ABB RobotStudio station: PR15CintasInteligentesEnunciado.rspag

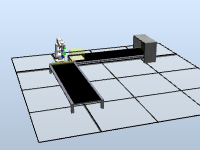
--- station ---
Station Station (saved by RobotStudio 6.5.7392.129)
Controller Sistema3
  mechanical unit ROB_1: IRB120_3_58__01, 6 joints, base frame (0, 0, 0) mm
Layout (positions relative to the parent item):
  - IRB120_3_58__01 [mechanism, from Robots\IRB120_3_58_G_01.rslib] at (0, 0, 0) mm; joint values [0, 0, 0, 0, 1.5708, 0] (rad or m)
  - SC_VentosaD50 [smart component] at (302, 0, 558) mm, rotated rx 180 ry 0 rz 180 deg
      signals: DI ElecVenturiVacio, DO ContactoVacuostato
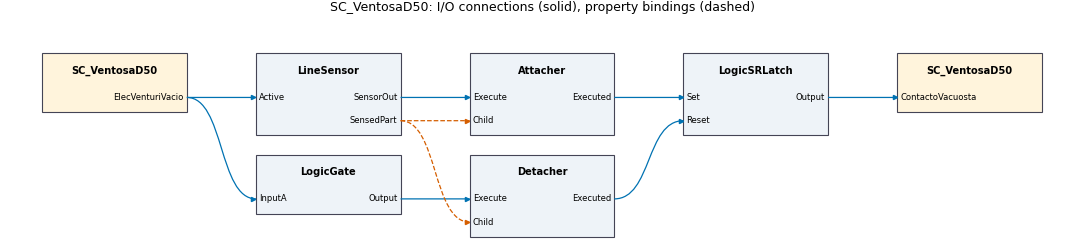
      connections:
        SC_VentosaD50.ElecVenturiVacio -> LineSensor.Active
        LineSensor.SensorOut -> Attacher.Execute
        Attacher.Executed -> LogicSRLatch.Set
        LogicSRLatch.Output -> SC_VentosaD50.ContactoVacuostato
        SC_VentosaD50.ElecVenturiVacio -> LogicGate.InputA
        LogicGate.Output -> Detacher.Execute
        Detacher.Executed -> LogicSRLatch.Reset
        LineSensor.SensedPart => Attacher.Child
        LineSensor.SensedPart => Detacher.Child
    - ToolVentosaD50 [mechanism] at (0, 0, 0) mm
        TCP TCP_ToolVentosaD50 at (0, 0, 129.5) mm
        links: VentosaCompletaD50
    - Attacher [smart component, from Components\Attacher.rslib]
        properties: Parent=ToolVentosaD50; Flange=0; Child=(none); Mount=false; Offset=[0 0 0]; Orientation=[0 0 0]
    - Detacher [smart component, from Components\Detacher.rslib]
        properties: Child=(none); KeepPosition=true
    - LineSensor [smart component, from Components\LineSensor.rslib] at (0, 0, 126) mm
        properties: Start=[0 0 0]; End=[0 0 0.015]; Radius=0.001; SensedPart=(none); SensedPoint=[3.0517578125E-08 0.427339996337891 0.290037750244141]
      - _sensorPart_ [part]
    - LogicGate [smart component, from Components\LogicGate.rslib]
        properties: Operator=NOT; Delay=0
    - LogicSRLatch [smart component, from Components\LogicSRLatch.rslib]
  - SC_CintaTransportadoraAlimentador [smart component] at (250, -300, 0) mm
      signals: DI diMotorCinta, DO doSensorCajas
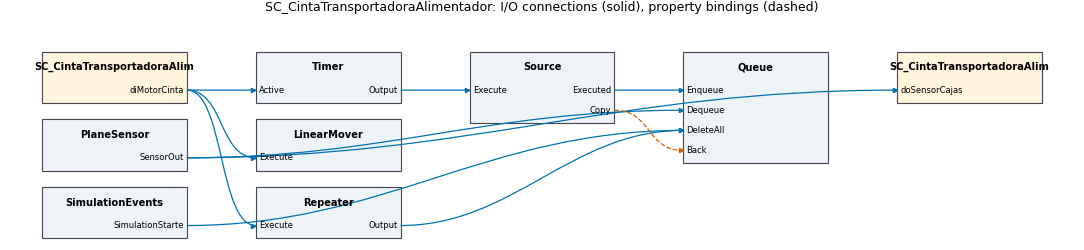
      connections:
        SC_CintaTransportadoraAlimentador.diMotorCinta -> Timer.Active
        SC_CintaTransportadoraAlimentador.diMotorCinta -> LinearMover.Execute
        Timer.Output -> Source.Execute
        Source.Executed -> Queue.Enqueue
        PlaneSensor.SensorOut -> Queue.Dequeue
        PlaneSensor.SensorOut -> SC_CintaTransportadoraAlimentador.doSensorCajas
        SC_CintaTransportadoraAlimentador.diMotorCinta -> Repeater.Execute
        Repeater.Output -> Queue.DeleteAll
        SimulationEvents.SimulationStarted -> Queue.DeleteAll
        Source.Copy => Queue.Back
    - CajaMaster [part] at (77.34, -250.57, -0.86) mm
    - CintaTransportadora [part]
    - Source [smart component, from Components\Source.rslib]
        properties: Source=CajaMaster; Copy=(none); Parent=(none); Position=[1.8 0.2 0.19]; Orientation=[0 0 0]; Transient=true; PhysicsBehavior=0
    - Queue [smart component, from Components\Queue.rslib]
        properties: Back=(none); Front=(none); Queue={a177aae2-69c8-43c3-9635-1530efa5db72}; NumberOfObjects=1
    - LinearMover [smart component, from Components\LinearMover.rslib]
        properties: Object=Queue; Direction=[-2.5 0 0]; Speed=0.5; Reference=Local; ReferenceObject=(none)
    - PlaneSensor [smart component, from Components\PlaneSensor.rslib]
        properties: Origin=[0.077626 0.55 0.19]; Axis1=[0 -0.5 0]; Axis2=[0 0 0.1]; SensedPart=(none)
      - _sensorPart_ [part]
    - Timer [smart component, from Components\Timer.rslib]
        properties: StartTime=0; Interval=2; Repeat=true; CurrentTime=11.688
    - SimulationEvents [smart component, from Components\SimulationEvents.rslib]
  - SC_CintaTransportadoraAlmacen [smart component] at (300, 250, 0) mm, rotated rx 0 ry 0 rz 90 deg
      signals: DI diConectarCinta, DO doObjetoAlmacenado
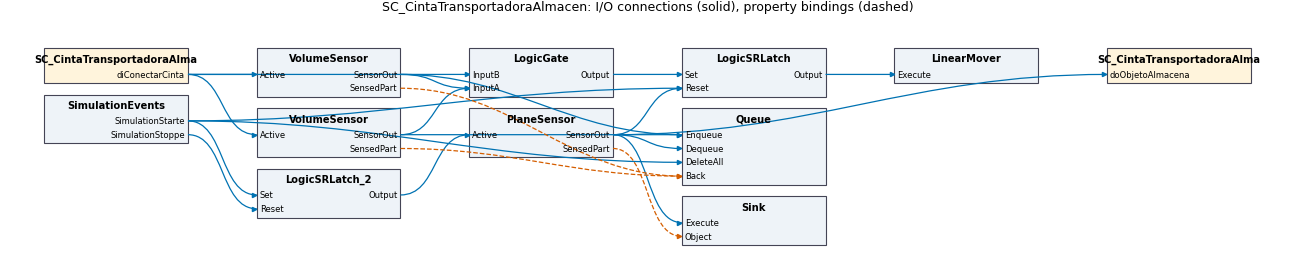
      connections:
        SC_CintaTransportadoraAlmacen.diConectarCinta -> VolumeSensor.Active
        VolumeSensor.SensorOut -> Queue.Enqueue
        PlaneSensor.SensorOut -> Sink.Execute
        PlaneSensor.SensorOut -> Queue.Dequeue
        PlaneSensor.SensorOut -> SC_CintaTransportadoraAlmacen.doObjetoAlmacenado
        SC_CintaTransportadoraAlmacen.diConectarCinta -> LogicGate.InputB
        VolumeSensor.SensorOut -> LogicGate.InputA
        LogicGate.Output -> LogicSRLatch.Set
        PlaneSensor.SensorOut -> LogicSRLatch.Reset
        SimulationEvents.SimulationStarted -> LogicSRLatch.Reset
        LogicSRLatch.Output -> LinearMover.Execute
        SimulationEvents.SimulationStarted -> Queue.DeleteAll
        SC_CintaTransportadoraAlmacen.diConectarCinta -> VolumeSensor.Active
        VolumeSensor.SensorOut -> Queue.Enqueue
        VolumeSensor.SensorOut -> LogicGate.InputA
        SimulationEvents.SimulationStarted -> LogicSRLatch_2.Set
        SimulationEvents.SimulationStopped -> LogicSRLatch_2.Reset
        LogicSRLatch_2.Output -> PlaneSensor.Active
        PlaneSensor.SensedPart => Sink.Object
        VolumeSensor.SensedPart => Queue.Back
        VolumeSensor.SensedPart => Queue.Back
    - CintaTransportadoraAlmacen [part]
    - PlaneSensor [smart component, from Components\PlaneSensor.rslib]
        properties: Origin=[1.82 0.05 0.19]; Axis1=[0 0.5 0]; Axis2=[0 0 0.1]; SensedPart=(none)
      - _sensorPart_ [part]
    - LinearMover [smart component, from Components\LinearMover.rslib]
        properties: Object=Queue; Direction=[0 2 0]; Speed=0.5; Reference=Local; ReferenceObject=(none)
    - Sink [smart component, from Components\Sink.rslib]
        properties: Object=(none)
    - Queue [smart component, from Components\Queue.rslib]
        properties: Back=(none); Front=(none); Queue={25e99bec-0593-4a2f-b814-1a7576071e65};{98dbe19b-009c-41f3-806d-1d9e1b097d57};{b6cd6502-60c9-460c-b551-ac68a1bc7dd4};{e8b803b3-ce63-45f2-91e8-1e93a9acf6e2}; NumberOfObjects=1
    - LogicGate [smart component, from Components\LogicGate.rslib]
        properties: Operator=AND; Delay=2
    - LogicSRLatch [smart component, from Components\LogicSRLatch.rslib]
    - SimulationEvents [smart component, from Components\SimulationEvents.rslib]
    - VolumeSensor [smart component, from Components\VolumeSensor.rslib]
        properties: CornerPoint=[0 0.15 0.191]; Orientation=[0 0 0]; Length=0.3; Width=0.3; Height=0.2; PartialHit=true; SensedPart=(none)
      - _sensorPart_ [part]
    - LogicSRLatch_2 [smart component, from Components\LogicSRLatch.rslib]
Attachment: SC_VentosaD50 is attached to IRB120_3_58__01 / Link6
Attachment: ToolVentosaD50 is attached to IRB120_3_58__01 / Link6
Targets, tools, work objects and paths stored in the station and not in the controller backup, written as RAPID:
! task T_ROB1
MODULE Module1
  CONST robtarget Inicio:=[[301.999967171,0,428.5],[-0.000000081,0,1,0],[-1,0,-1,0],[9E+09,9E+09,9E+09,9E+09,9E+09,9E+09]];
ENDMODULE


--- Backups/Sistema3/RAPID/TASK1/PROGMOD/CalibData.mod ---
MODULE CalibData
	PERS tooldata TCP_ToolVentosaD50:=[TRUE,[[0,0,129.5],[1,0,0,0]],[1,[0,0,1],[1,0,0,0],0,0,0]];
	TASK PERS wobjdata WoCinta:=[FALSE,TRUE,"",[[250,-300,0],[1,0,0,0]],[[0,0,0],[1,0,0,0]]];
ENDMODULE

--- Backups/Sistema3/RAPID/TASK1/PROGMOD/MainModule.mod ---
MODULE MainModule
    !***********************************************************
    !
    ! Módulo:  MainModule
    !
    ! Descripción:
    !   <Introduzca la descripción aquí>
    !
    ! Autor: Juan
    !
    ! Versión: 1.0
    !
    !***********************************************************


    !***********************************************************
    !
    ! Procedimiento Main
    !
    !   Este es el punto de entrada de su programa
    !
    !***********************************************************
    PROC main()



    ENDPROC
ENDMODULE

--- Backups/Sistema3/RAPID/TASK1/PROGMOD/Module1.mod ---
MODULE Module1

ENDMODULE

--- Backups/Sistema3/RAPID/TASK1/SYSMOD/LINKEDM.sys ---
%%%
  VERSION:1
  LANGUAGE:ENGLISH
%%%

MODULE LINKEDM (SYSMODULE)

! FOLLOWER
!     Name of electronically linked follower axis used by operator at teach pendent.
      PERS string l_f_axis_name{5}       :=  ["",  "", "", "", ""];

!     Name of the mechanical unit for follower axis.
      PERS string l_f_mecunt_n{5}  :=  ["", "", "", "", ""];

!     Linked follower axis number in the mechanical unit (first axis in mech. unit is number 1).
      PERS num l_f_axis_no{5}      :=  [0,          0,   0,  0,  0];

! MASTER
!     Name of the mechanical unit for linked master axis.
      PERS string l_m_mecunt_n{5} :=  ["", "", "", "", ""];

!     Linked master axis number in the mechanical unit (first axis in mech. unit is number 1).
!     See axis number table in documentation for different master mechanical units.
      PERS num l_m_axis_no{5}     :=  [0,  0,  0,  0,  0];

! POSITION OFFSET
!     The increase of the allowed offset position between the master and follower
!     positions, used when starting AUTO mode. As soon as the offset is decreased
!     the old configurated parameter is used.
!     Example: 3 => the configurated value of allowed offset is increased 3 times.
      PERS num offset_ratio{5}       :=  [10,  10,   10,  10,  10];

! SPEED RATIO
!     Speed_ratio used in AUTO and JOG modes [ very_slow   slow    normal    fast]
!     Value 1 = max allowed manual speed.
      CONST num speed_ratio {20}      := [0.01, 0.01, 0.01, 0.01, 0.01,
                                          0.05, 0.05, 0.05, 0.05, 0.05,
                                          0.20, 0.20, 0.20, 0.20, 0.20,
                                          1.00, 1.00, 1.00, 1.00, 1.00];

! STEP SIZE
!     Displacement position used in JOG mode for each activation of positive or
!     negative movement.                  [very_short    short   normal   long]
!     Unit degees or meter.
      CONST num displacement {20}     := [0.001, 0.001, 0.001, 0.001, 0.001,
                                          0.005, 0.005, 0.005, 0.005, 0.005,
                                          0.020, 0.020, 0.020, 0.020, 0.020,
                                          0.100, 0.100, 0.100, 0.100, 0.100];


!-------------------------------------------------------------
 PROC Linked_m ()
      Linked_m_exe ;
 ENDPROC
ENDMODULE

--- Backups/Sistema3/SYSPAR/EIO.cfg ---
EIO:CFG_1.0:6:1::
#
INDUSTRIAL_NETWORK:

      -Name "PROFINET" -Connection "PROFINET Network"\
      -Label "PROFINET Controller/Device Network" -StationName ""
#
PROFINET_INTERNAL_DEVICE:

      -Name "PN_Internal_Device" -VendorName "ABB Robotics"\
      -ProductName "PROFINET Internal Device"
#
EIO_SIGNAL:

      -Name "DI_1" -SignalType "DI" -Device "PN_Internal_Device"\
      -Label "Entrada digital 1" -DeviceMap "128"

      -Name "DI_2" -SignalType "DI" -Device "PN_Internal_Device"\
      -Label "Entrada digital 2" -DeviceMap "129"

      -Name "DI_3" -SignalType "DI" -Device "PN_Internal_Device"\
      -Label "Entrada digital 3" -DeviceMap "130"

      -Name "DI_4" -SignalType "DI" -Device "PN_Internal_Device"\
      -Label "Entrada digital 4" -DeviceMap "131"

      -Name "DI_5" -SignalType "DI" -Device "PN_Internal_Device"\
      -Label "Entrada digital 5" -DeviceMap "132"

      -Name "DI_6" -SignalType "DI" -Device "PN_Internal_Device"\
      -Label "Entrada digital 6" -DeviceMap "133"

      -Name "DI_8" -SignalType "DI" -Device "PN_Internal_Device"\
      -Label "Entrada digital 8" -DeviceMap "135"

      -Name "DO_1" -SignalType "DO" -Device "PN_Internal_Device"\
      -Label "Salida digital 1" -DeviceMap "136"

      -Name "DO_2" -SignalType "DO" -Device "PN_Internal_Device"\
      -Label "Salida digital 2" -DeviceMap "137"

      -Name "DO_3" -SignalType "DO" -Device "PN_Internal_Device"\
      -Label "Salida digital 3" -DeviceMap "138"

      -Name "DO_4" -SignalType "DO" -Device "PN_Internal_Device"\
      -Label "Salida digital 4" -DeviceMap "139"

      -Name "DO_5" -SignalType "DO" -Device "PN_Internal_Device"\
      -Label "Salida digital 5" -DeviceMap "140"

      -Name "DO_6" -SignalType "DO" -Device "PN_Internal_Device"\
      -Label "Salida digital 6" -DeviceMap "141"

      -Name "DI_7" -SignalType "DI" -Device "PN_Internal_Device"\
      -Label "Entrada digital 7" -DeviceMap "134"

      -Name "DO_7" -SignalType "DO" -Device "PN_Internal_Device"\
      -Label "Salida digital 7" -DeviceMap "142"

      -Name "DO_8" -SignalType "DO" -Device "PN_Internal_Device"\
      -Label "Salida digital 8" -DeviceMap "143"
